Fanuc KAREL source: kt00485.KL

-- PROVISIONAL review KL for V940-1; original PC SHA256 c1393ba5bd0841b770255e3b4a84a9e5cbf9b5bb69e99aa6b5de74db30d90d12
-- Incomplete behavior may be omitted. Consult companion uncertainty JSON. Do not deploy.
PROGRAM KT00485
%NOLOCKGROUP
-- UNRESOLVED_DECL P1 type=000101
-- UNRESOLVED_DECL P2 type=000106
-- UNRESOLVED_DECL OUT type=000102
BEGIN
  -- V9_ZERO_TABLE_METADATA_HINT layout=0001; no indexed target words; source/name/runtime held
  -- UNRESOLVED_PC offsets 5-20; opcodes 2E,22,32,35
  -- UNRESOLVED_PC offsets 25-59; opcodes 49,49,7E,60,7E,4A
  -- UNRESOLVED_PC offsets 64-68; opcodes 7F
END KT00485
